Staubli VAL3: OnEvent13.pgx

program OnEvent13()
begin
  //-----------------------------------------------------------------------
  //Header begin
  //LasMAN3.7
  //Description of program
  //
  //Input parameters
  //
  //Output paramaters
  //Example
  //  call OnEvent1()
  //History
  //  Creation : 2013-06-23  y.ye@staubli.com
  //Header end
  //-----------------------------------------------------------------------
  resetMotion()
  call Teach:TeachProduct()
  DataBase:nInterfaceType=9
end
